FUNCTION FC_WithinRange : BOOL		// Checks if the specified value is within the target range, returns TRUE if within range, FALSE otherwise
VAR_INPUT
	iValue:			LREAL;		// Value to be checked
	iTarget:		LREAL;		// Target value
	iRange:			LREAL;		// This value is allowed below and above
END_VAR
VAR
	minValue:	LREAL;
	maxValue:	LREAL;
END_VAR

minValue := iTarget - iRange;
maxValue := iTarget + iRange;
FC_WithinRange := (iValue >= minValue) AND (iValue <= maxValue);

END_FUNCTION

(* stored: Version 1.1.0.1, ProductVersion 3.1.4026.18
   POU FC_WithinRange: Id {3901acfa-0a9d-40e4-a9dd-0c971f87a8ab}, SpecialFunc None *)
